INTERFACE I_PixelReader

PROPERTY PUBLIC Value : Reference to TcVnVector4_LREAL
GET
END_GET
END_PROPERTY

END_INTERFACE

(* stored: Version 1.1.0.1
   Itf I_PixelReader: Id {4834e65f-15d0-4adc-83a4-1dcb60389701}
   Property Value: Id {10ca9ecb-eded-4dfa-a3b7-e67bfb0d4509}
   Get Get: Id {b931c3ef-1860-4dd0-b61e-86b07b841634} *)
